// Mitsubishi GX Works2 project: may_dap_FX1S   PLC: FX3S

PROGRAM MAIN
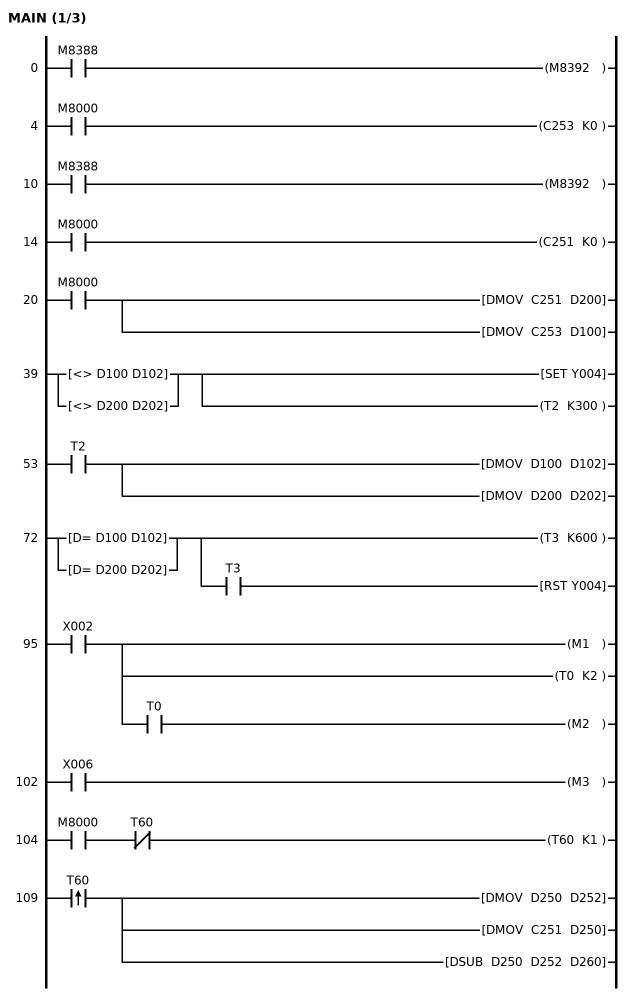
0     LD      M8388
      OUT     M8392
4     LD      M8000
      OUT     C253 K0
10    LD      M8388
      OUT     M8392
14    LD      M8000
      OUT     C251 K0
20    LD      M8000
      DMOV    C251 D200
      DMOV    C253 D100
39    LD<>    D100 D102
      OR<>    D200 D202
      SET     Y004
      OUT     T2 K300
53    LD      T2
      DMOV    D100 D102
      DMOV    D200 D202
72    LDD=    D100 D102
      ORD=    D200 D202
      OUT     T3 K600
      AND     T3
      RST     Y004
95    LD      X002
      OUT     M1
      OUT     T0 K2
      AND     T0
      OUT     M2
102   LD      X006
      OUT     M3
104   LD      M8000
      ANI     T60
      OUT     T60 K1
109   LDP     T60
      DMOV    D250 D252
      DMOV    C251 D250
      DSUB    D250 D252 D260
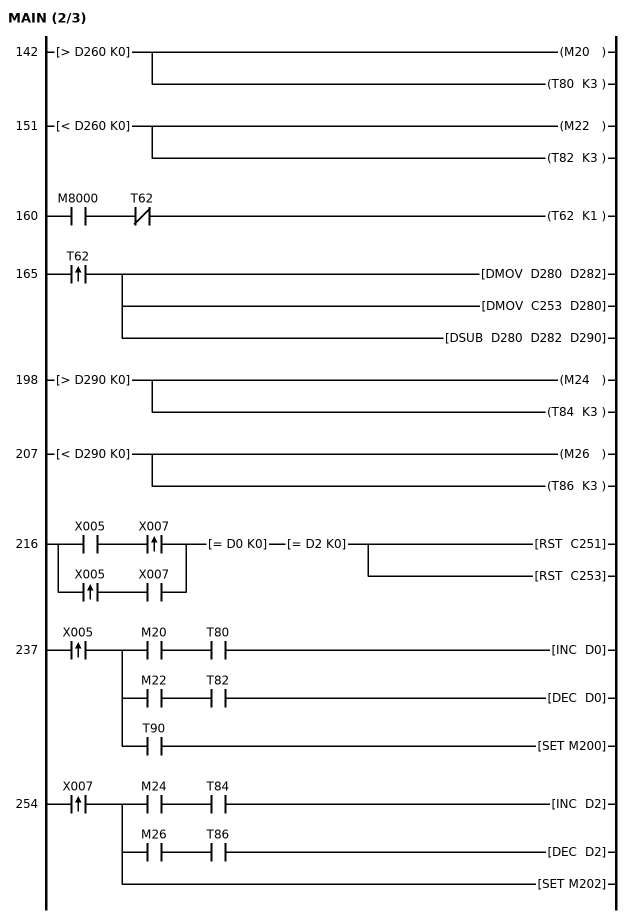
142   LD>     D260 K0
      OUT     M20
      OUT     T80 K3
151   LD<     D260 K0
      OUT     M22
      OUT     T82 K3
160   LD      M8000
      ANI     T62
      OUT     T62 K1
165   LDP     T62
      DMOV    D280 D282
      DMOV    C253 D280
      DSUB    D280 D282 D290
198   LD>     D290 K0
      OUT     M24
      OUT     T84 K3
207   LD<     D290 K0
      OUT     M26
      OUT     T86 K3
216   LD      X005
      ANDP    X007
      LDP     X005
      AND     X007
      ORB
      AND=    D0 K0
      AND=    D2 K0
      RST     C251
      RST     C253
237   LDP     X005
      MPS
      AND     M20
      AND     T80
      INC     D0
      MRD
      AND     M22
      AND     T82
      DEC     D0
      MPP
      AND     T90
      SET     M200
254   LDP     X007
      MPS
      AND     M24
      AND     T84
      INC     D2
      MRD
      AND     M26
      AND     T86
      DEC     D2
      MPP
      SET     M202
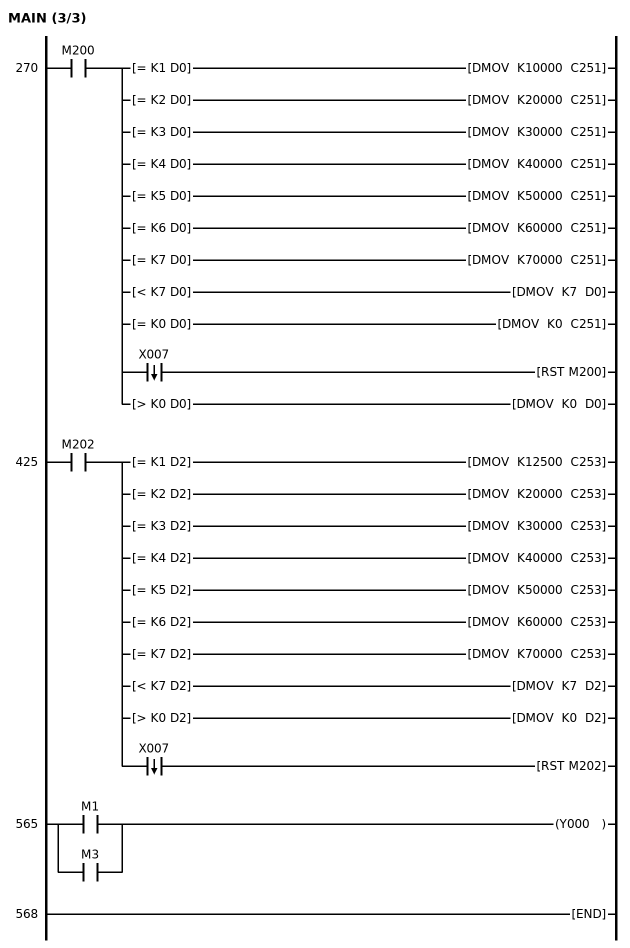
270   LD      M200
      MPS
      AND=    K1 D0
      DMOV    K10000 C251
      MRD
      AND=    K2 D0
      DMOV    K20000 C251
      MRD
      AND=    K3 D0
      DMOV    K30000 C251
      MRD
      AND=    K4 D0
      DMOV    K40000 C251
      MRD
      AND=    K5 D0
      DMOV    K50000 C251
      MRD
      AND=    K6 D0
      DMOV    K60000 C251
      MRD
      AND=    K7 D0
      DMOV    K70000 C251
      MRD
      AND<    K7 D0
      DMOV    K7 D0
      MRD
      AND=    K0 D0
      DMOV    K0 C251
      MRD
      ANDF    X007
      RST     M200
      MPP
      AND>    K0 D0
      DMOV    K0 D0
425   LD      M202
      MPS
      AND=    K1 D2
      DMOV    K12500 C253
      MRD
      AND=    K2 D2
      DMOV    K20000 C253
      MRD
      AND=    K3 D2
      DMOV    K30000 C253
      MRD
      AND=    K4 D2
      DMOV    K40000 C253
      MRD
      AND=    K5 D2
      DMOV    K50000 C253
      MRD
      AND=    K6 D2
      DMOV    K60000 C253
      MRD
      AND=    K7 D2
      DMOV    K70000 C253
      MRD
      AND<    K7 D2
      DMOV    K7 D2
      MRD
      AND>    K0 D2
      DMOV    K0 D2
      MPP
      ANDF    X007
      RST     M202
565   LD      M1
      OR      M3
      OUT     Y000
568   END
END_PROGRAM
